PROGRAM pouS3Prompts
VAR
	


idbMsgPrompt: FB_CheckMessageBounds;
END_VAR

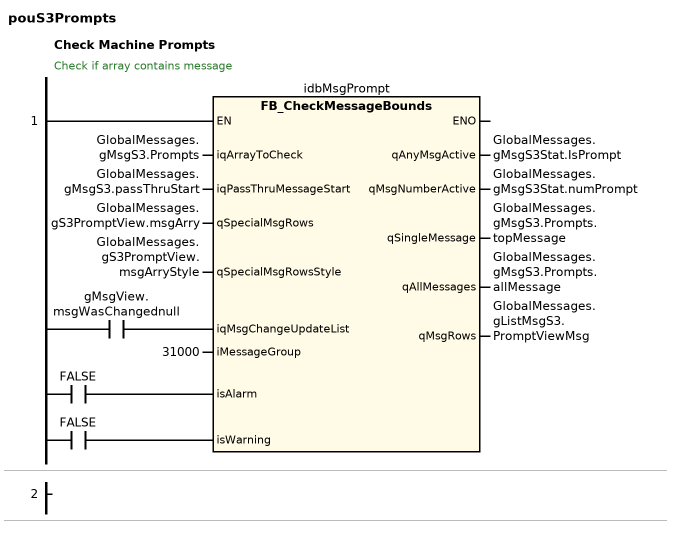
// NETWORK 1: Check Machine Prompts
// Check if array contains message
idbMsgPrompt(
    iqArrayToCheck := GlobalMessages.gMsgS3.Prompts,
    iqPassThruMessageStart := GlobalMessages.gMsgS3.passThruStart,
    qSpecialMsgRows := GlobalMessages.gS3PromptView.msgArry,
    qSpecialMsgRowsStyle := GlobalMessages.gS3PromptView.msgArryStyle,
    iqMsgChangeUpdateList := gMsgView.msgWasChangednull,
    iMessageGroup := 31000,
    isAlarm := FALSE,
    isWarning := FALSE,
    qAnyMsgActive => GlobalMessages.gMsgS3Stat.IsPrompt,
    qMsgNumberActive => GlobalMessages.gMsgS3Stat.numPrompt,
    qSingleMessage => GlobalMessages.gMsgS3.Prompts.topMessage,
    qAllMessages => GlobalMessages.gMsgS3.Prompts.allMessage,
    qMsgRows => GlobalMessages.gListMsgS3.PromptViewMsg); // FB_CheckMessageBounds

// NETWORK 2

END_PROGRAM

(* stored: Version 1.1.0.1, ProductVersion 3.1.4024.11
   POU pouS3Prompts: Id {0a6de161-75b2-4807-ac03-9dc22597f730}, SpecialFunc None *)
